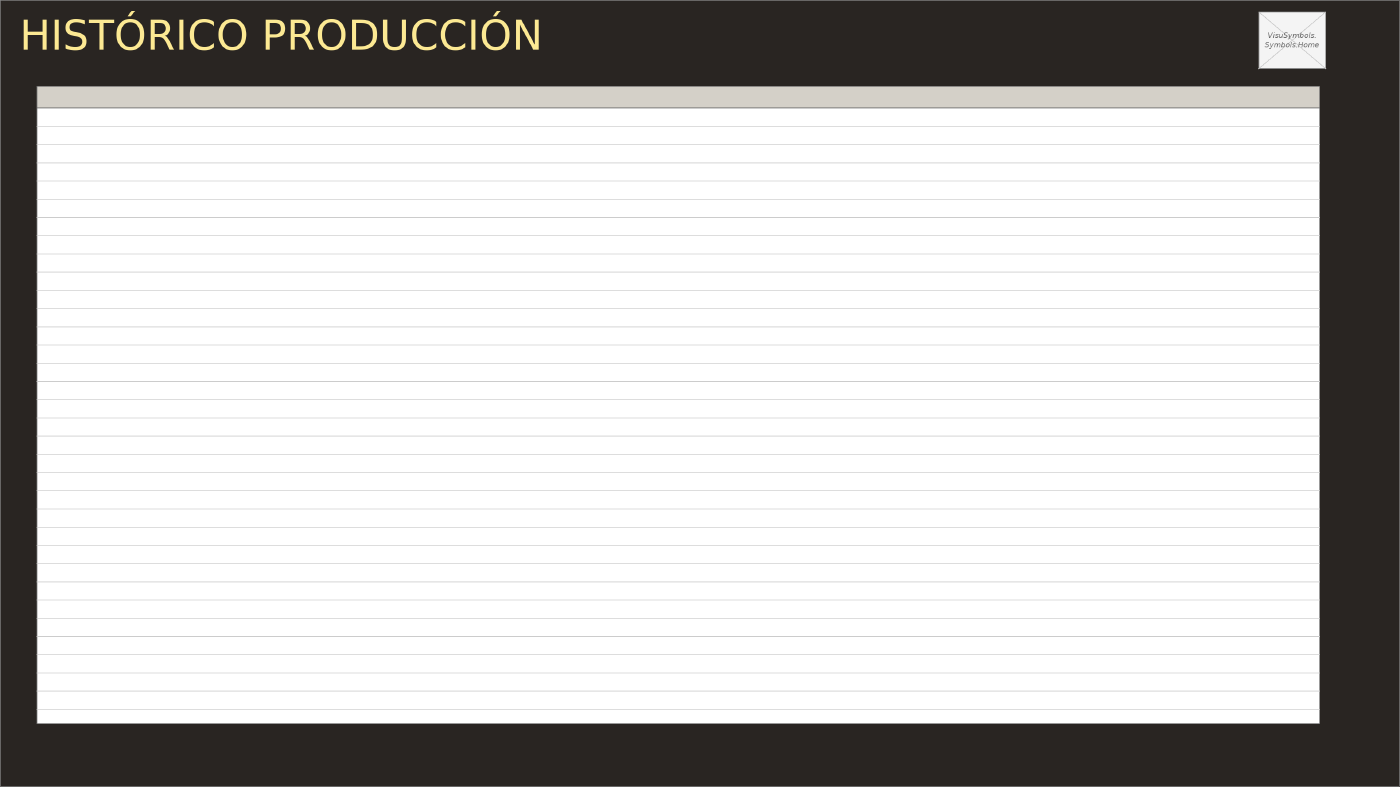
VISUALIZATION HistTablaTablas_Ch2  // 1920x1080
    Image (1726,16 92x78), image: VisuSymbols.Symbols.Home
        OnMouseClick: change screen: Home_CortH2
    Table (50,118 1760x875), data array: RegistroLocalDataBase.aHistoricStrTablasCH2
        p3854506369: RegistroLocalDataBase.aHistoricStrTablasCH2[INDEX].ID
        p1892666644: RegistroLocalDataBase.aHistoricStrTablasCH2[INDEX].Fecha
        p338671338: RegistroLocalDataBase.aHistoricStrTablasCH2[INDEX].Modelo
        p2170511999: RegistroLocalDataBase.aHistoricStrTablasCH2[INDEX].Formato
        p3723444502: RegistroLocalDataBase.aHistoricStrTablasCH2[INDEX].Espesor
        p1218418051: RegistroLocalDataBase.aHistoricStrTablasCH2[INDEX].Maquina
        p746581629: RegistroLocalDataBase.aHistoricStrTablasCH2[INDEX].Cont_Piezas
        p3104783080: RegistroLocalDataBase.aHistoricStrTablasCH2[INDEX].t_Entre_Piez_Ftc
        p2501879983: RegistroLocalDataBase.aHistoricStrTablasCH2[INDEX].S_Justi_Paro_Ftc
        p1757482276: Numero de tablas
        p4088588272: Tiempo entre tablas
        p2243050616: Justificación del paro
    Label (24,16 669x64), "HISTÓRICO PRODUCCIÓN"
END_VISUALIZATION

(* stored: Version 1.1.0.1, ProductVersion 3.1.4024.12
   Visu HistTablaTablas_Ch2: Id {169d72ac-5c2b-4084-979b-fd36a443784b} *)
